# EPICS substitutions: siteApps/siemensPLC/iocBoot/iocs7Modbus/StepMTst.substitutions
# These are the Digital Coil inputs with StepMTst
file "db/bi_bit.template" { pattern
{P,           R,         PORT,             OFFSET,   ZNAM,   ONAM,  ZSV,       OSV,    SCAN}
{STEP:,    CInB0,     Step_Motor_CIn_Bit,     0,     Low,    High,  NO_ALARM,  MAJOR,  "I/O Intr"}
{STEP:,    CInB1,     Step_Motor_CIn_Bit,     1,     Low,    High,  NO_ALARM,  MAJOR,  "I/O Intr"}
{STEP:,    CInB2,     Step_Motor_CIn_Bit,     2,     Low,    High,  NO_ALARM,  MAJOR,  "I/O Intr"}
{STEP:,    CInB3,     Step_Motor_CIn_Bit,     3,     Low,    High,  NO_ALARM,  MAJOR,  "I/O Intr"}
{STEP:,    CInB4,     Step_Motor_CIn_Bit,     4,     Low,    High,  NO_ALARM,  MAJOR,  "I/O Intr"}
{STEP:,    CInB5,     Step_Motor_CIn_Bit,     5,     Low,    High,  NO_ALARM,  MAJOR,  "I/O Intr"}
{STEP:,    CInB6,     Step_Motor_CIn_Bit,     6,     Low,    High,  NO_ALARM,  MAJOR,  "I/O Intr"}
{STEP:,    CInB7,     Step_Motor_CIn_Bit,     7,     Low,    High,  NO_ALARM,  MAJOR,  "I/O Intr"}
}
